// SIMATIC S7-200 project (STEP 7-Micro/WIN), CPU 226 CN REL 02.01

ORGANIZATION_BLOCK OB_1:OB1
TITLE=Ver41 add  weekly  timer  to  PLC , and  Clean Claw Pump check ;  PC program use  Ver34 edition  or  higher edition .
// Ver42  shifting  change ,  
// Ver43  add 喷雾提前结束(20060822) , PC Program 使用Ver35或以上版本
// Ver43  communication format  change  , PC程序使用Ver21或以上版本
// ver44  PC程序使用Ver21或以上版本
// Ver45  增加热补偿和PCB阻塞报警,PC程序使用Ver22或以上版本
// Ver46  增加付款条件自锁功能
// Ver47  完善喷雾（可提前或延时结束）
// ver48  细化运输模拟量参数
BEGIN
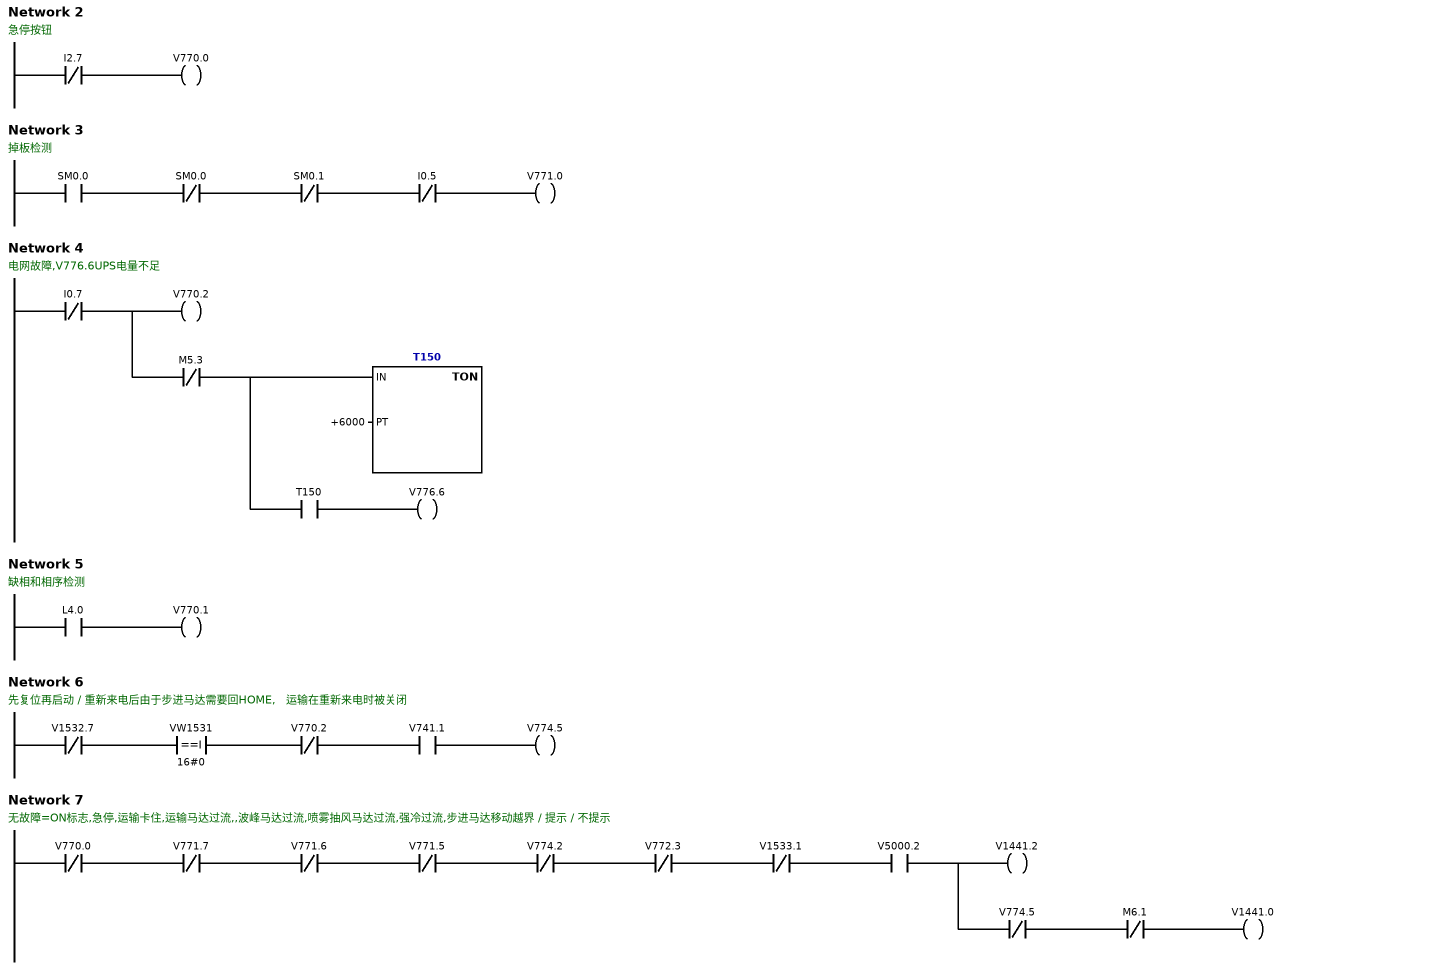
Network 2
// 急停按钮
LDN    I2.7
=      V770.0
Network 3
// 掉板检测
LD     SM0.0
AN     SM0.0
AN     SM0.1
AN     I0.5
=      V771.0
Network 4
// 电网故障,V776.6UPS电量不足
LDN    I0.7
=      V770.2
AN     M5.3
TON    T150, +6000
A      T150
=      V776.6
Network 5
// 缺相和相序检测
LD     L4.0
=      V770.1
Network 6
// 先复位再启动
// 重新来电后由于步进马达需要回HOME,   运输在重新来电时被关闭
LDN    V1532.7
AW=    VW1531, 16#0
AN     V770.2
A      V741.1
=      V774.5
Network 7
// 无故障=ON标志,急停,运输卡住,运输马达过流,,波峰马达过流,喷雾抽风马达过流,强冷过流,步进马达移动越界
// 提示
// 不提示
LDN    V770.0
AN     V771.7
AN     V771.6
AN     V771.5
AN     V774.2
AN     V772.3
AN     V1533.1
A      V5000.2
=      V1441.2
AN     V774.5
AN     M6.1
=      V1441.0
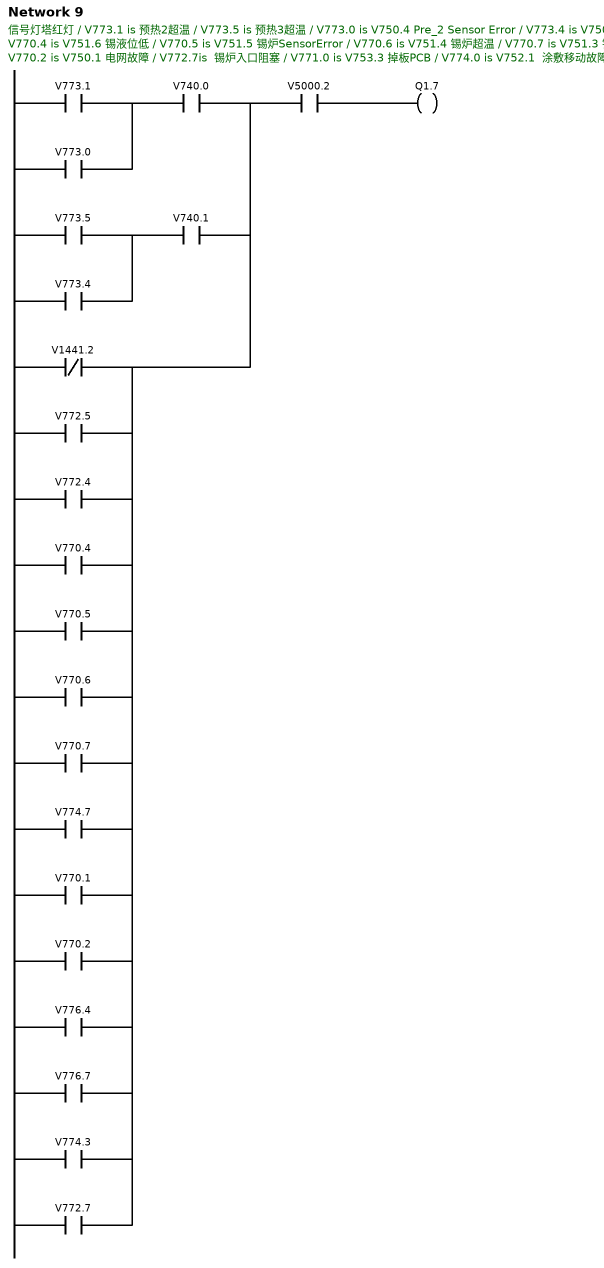
Network 9
// 信号灯塔红灯
// V773.1 is 预热2超温
// V773.5 is 预热3超温
// V773.0 is V750.4 Pre_2 Sensor Error
// V773.4 is V750.5 Pre_3 Sensor Error
// V772.5 is 预热1超温
// V772.4 is V750.3 Pre_1 Sensor Error
// 
// V770.4 is V751.6 锡液位低
// V770.5 is V751.5 锡炉SensorError
// V770.6 is V751.4 锡炉超温
// V770.7 is V751.3 锡炉参数错误
// V774.7 is V751.7  防止锡炉超温控制器
// 
// V770.1 is V750.0 电网缺相/相序错误
// V770.2 is V750.1 电网故障
// V772.7is  锡炉入口阻塞
// V771.0 is V753.3 掉板PCB
// V774.0 is V752.1  涂敷移动故障
// V776.4 is V752.3  助焊剂缺少
// V776.7 is V752.5  Clean Claw Low Limit
// V1533.1 is V752.4 步进马达移动故障
// V774.3 is V752.6 助焊剂添加故障
LD     V773.1
O      V773.0
A      V740.0
LD     V773.5
O      V773.4
A      V740.1
OLD
LDN    V1441.2
O      V772.5
O      V772.4
O      V770.4
O      V770.5
O      V770.6
O      V770.7
O      V774.7
O      V770.1
O      V770.2
O      V776.4
O      V776.7
O      V774.3
O      V772.7
OLD
A      V5000.2
=      Q1.7
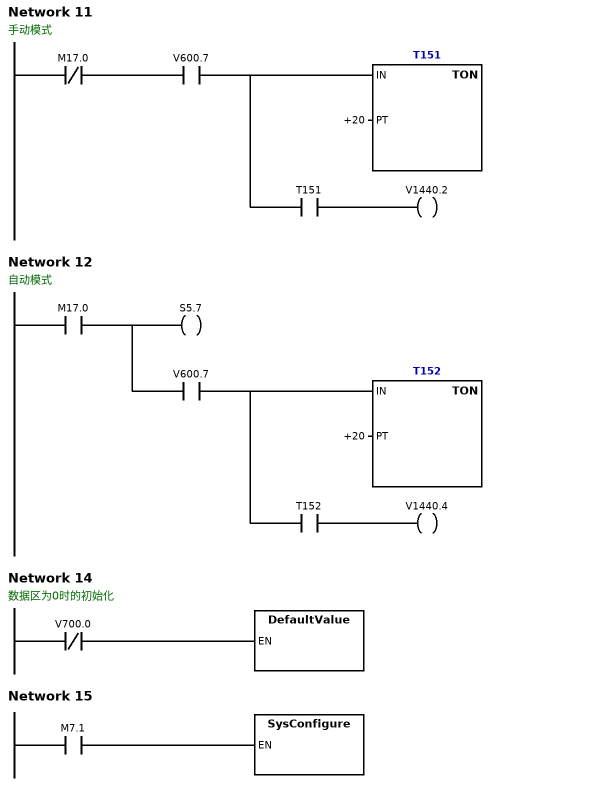
Network 11
// 手动模式
LDN    M17.0
A      V600.7
TON    T151, +20
A      T151
=      V1440.2
Network 12
// 自动模式
LD     M17.0
=      S5.7
A      V600.7
TON    T152, +20
A      T152
=      V1440.4
Network 14
// 数据区为0时的初始化
LDN    V700.0
CALL   DefaultValue:SBR18
Network 15
LD     M7.1
CALL   SysConfigure:SBR29
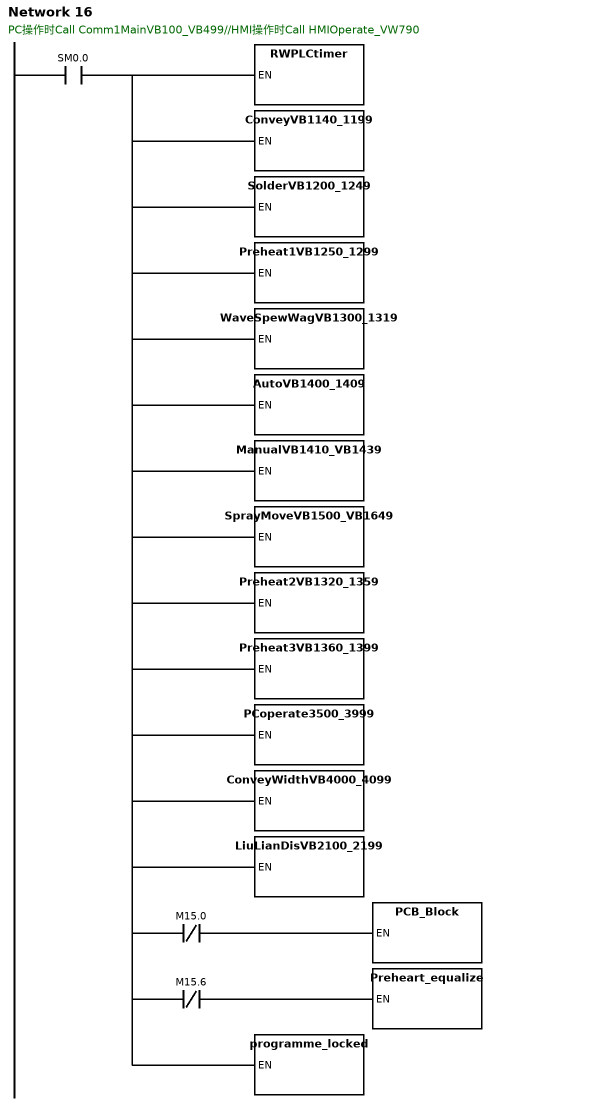
Network 16
// PC操作时Call Comm1MainVB100_VB499//HMI操作时Call HMIOperate_VW790
LD     SM0.0
LPS
CALL   RWPLCtimer:SBR1
CALL   ConveyVB1140_1199:SBR2
CALL   SolderVB1200_1249:SBR3
CALL   Preheat1VB1250_1299:SBR4
CALL   WaveSpewWagVB1300_1319:SBR5
CALL   AutoVB1400_1409:SBR8
CALL   ManualVB1410_VB1439:SBR9
CALL   SprayMoveVB1500_VB1649:SBR10
CALL   Preheat2VB1320_1359:SBR6
CALL   Preheat3VB1360_1399:SBR7
CALL   PCoperate3500_3999:SBR17
CALL   ConveyWidthVB4000_4099:SBR16
CALL   LiuLianDisVB2100_2199:SBR11
AN     M15.0
CALL   PCB_Block:SBR45
LRD
AN     M15.6
CALL   Preheart_equalize:SBR34
LPP
CALL   programme_locked:SBR46
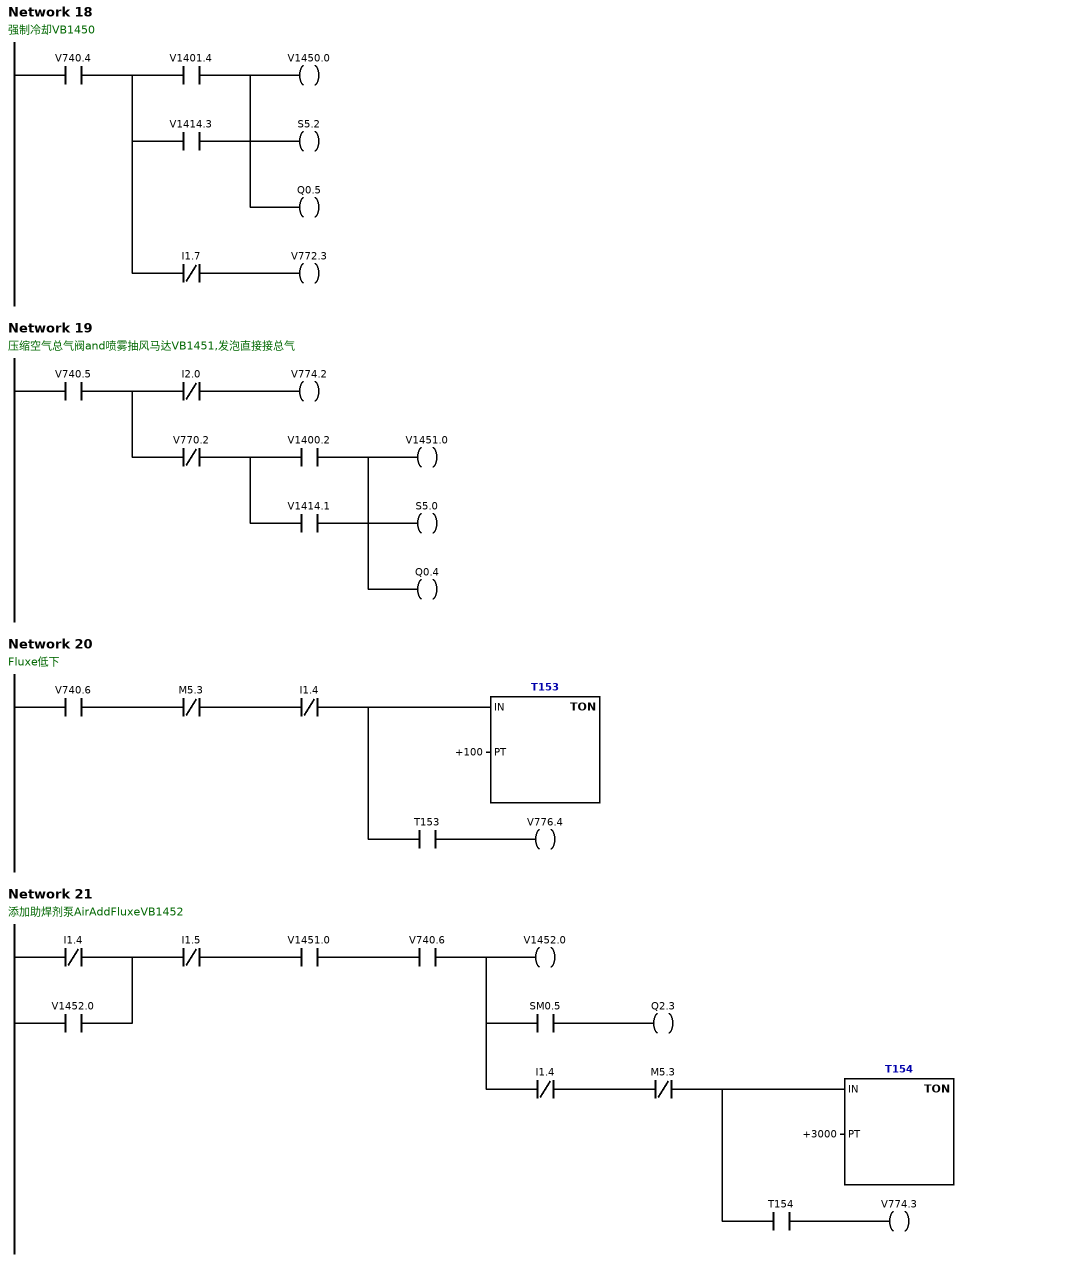
Network 18
// 强制冷却VB1450
LD     V740.4
LPS
LD     V1401.4
O      V1414.3
ALD
=      V1450.0
=      S5.2
=      Q0.5
LPP
AN     I1.7
=      V772.3
Network 19
// 压缩空气总气阀and喷雾抽风马达VB1451,发泡直接接总气
LD     V740.5
LPS
AN     I2.0
=      V774.2
LPP
AN     V770.2
LD     V1400.2
O      V1414.1
ALD
=      V1451.0
=      S5.0
=      Q0.4
Network 20
// Fluxe低下
LD     V740.6
AN     M5.3
AN     I1.4
TON    T153, +100
A      T153
=      V776.4
Network 21
// 添加助焊剂泵AirAddFluxeVB1452
LDN    I1.4
O      V1452.0
AN     I1.5
A      V1451.0
A      V740.6
LPS
=      V1452.0
A      SM0.5
=      Q2.3
LPP
AN     I1.4
AN     M5.3
TON    T154, +3000
A      T154
=      V774.3
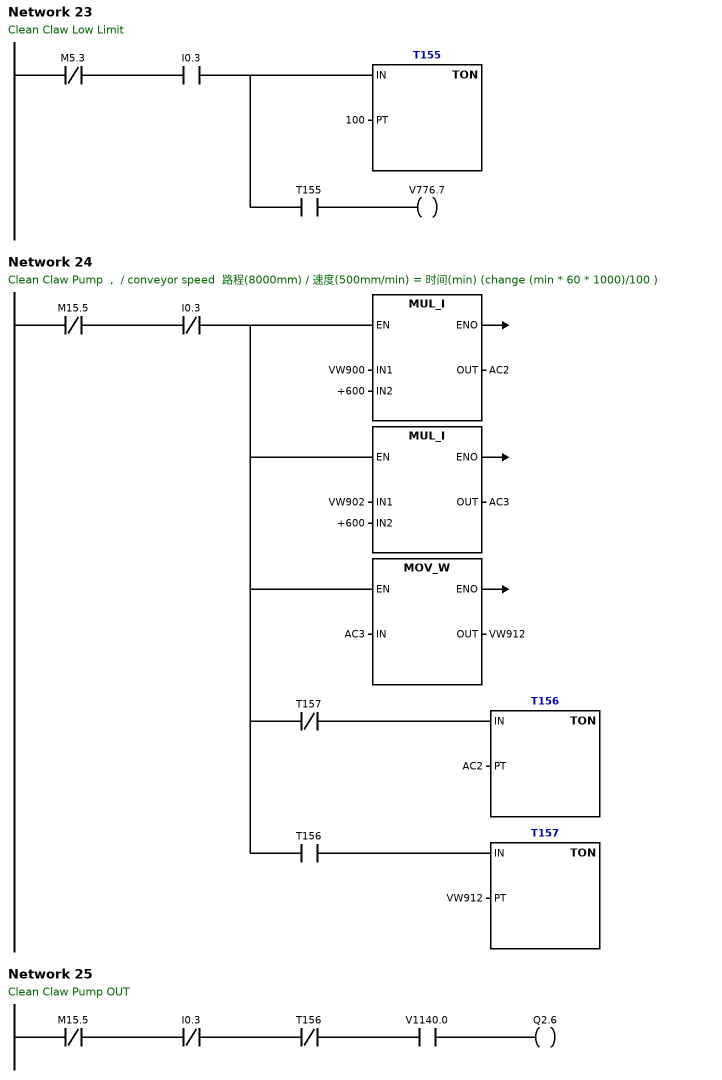
Network 23
// Clean Claw Low Limit
LDN    M5.3
A      I0.3
TON    T155, 100
A      T155
=      V776.7
Network 24
// Clean Claw Pump  , 
// conveyor speed  路程(8000mm) / 速度(500mm/min) = 时间(min) (change (min * 60 * 1000)/100 )
LDN    M15.5
AN     I0.3
LPS
MOVW   VW900, AC2
*I     +600, AC2
MOVW   VW902, AC3
*I     +600, AC3
MOVW   AC3, VW912
AN     T157
TON    T156, AC2
LPP
A      T156
TON    T157, VW912
Network 25
// Clean Claw Pump OUT
LDN    M15.5
AN     I0.3
AN     T156
A      V1140.0
=      Q2.6
END_ORGANIZATION_BLOCK

SUBROUTINE_BLOCK RWPLCtimer:SBR1
TITLE=
BEGIN
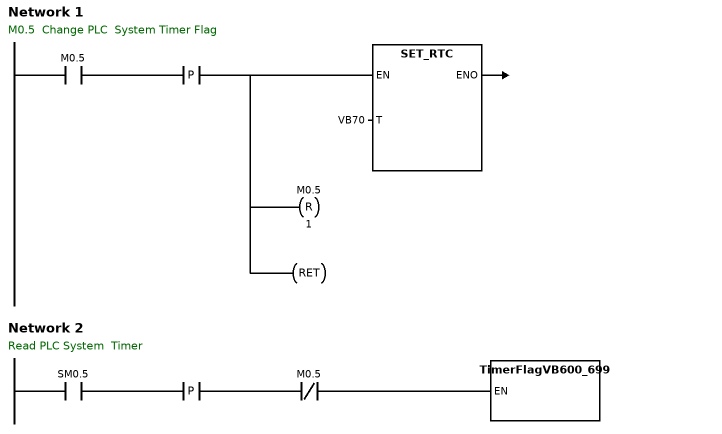
Network 1
//  M0.5  Change PLC  System Timer Flag
LD     M0.5
EU
TODW   VB70
R      M0.5, 1
CRET
Network 2 // 

// Read PLC System  Timer
LD     SM0.5
EU
AN     M0.5
CALL   TimerFlagVB600_699:SBR33
END_SUBROUTINE_BLOCK

SUBROUTINE_BLOCK ConveyVB1140_1199:SBR2
TITLE=
BEGIN
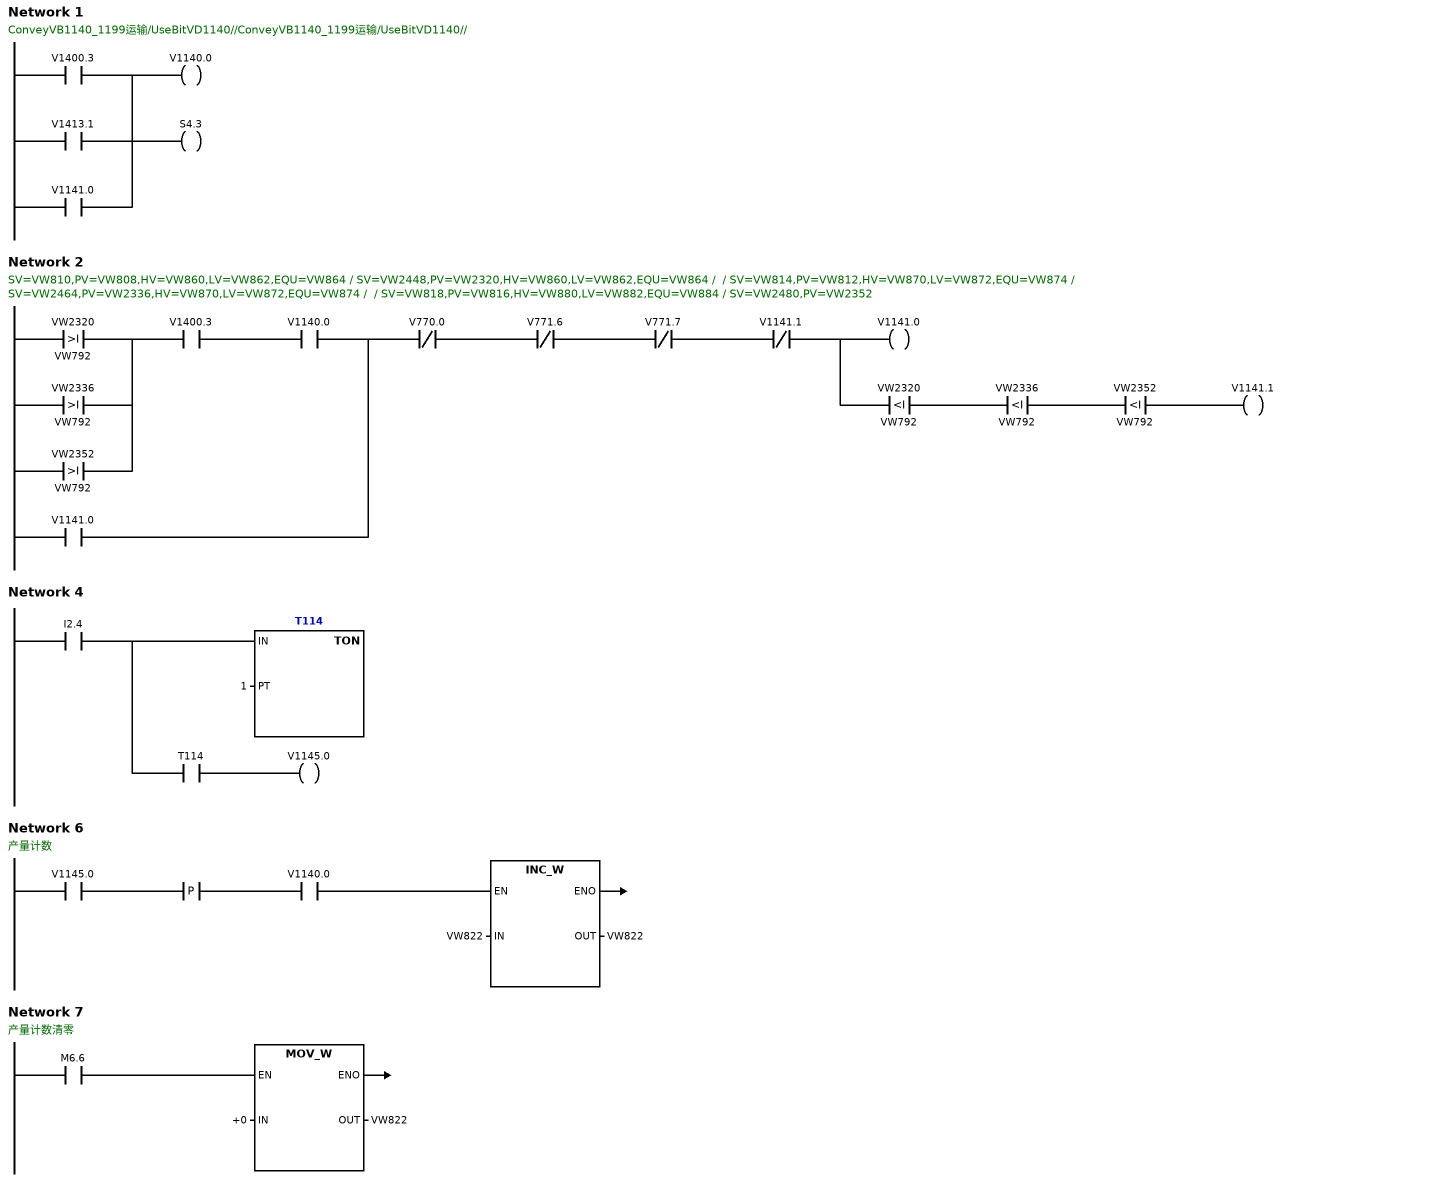
Network 1
// ConveyVB1140_1199运输/UseBitVD1140//ConveyVB1140_1199运输/UseBitVD1140//
LD     V1400.3
O      V1413.1
O      V1141.0
=      V1140.0
=      S4.3
Network 2
// SV=VW810,PV=VW808,HV=VW860,LV=VW862,EQU=VW864
// SV=VW2448,PV=VW2320,HV=VW860,LV=VW862,EQU=VW864
// 
// SV=VW814,PV=VW812,HV=VW870,LV=VW872,EQU=VW874
// SV=VW2464,PV=VW2336,HV=VW870,LV=VW872,EQU=VW874
// 
// SV=VW818,PV=VW816,HV=VW880,LV=VW882,EQU=VW884
// SV=VW2480,PV=VW2352
LDW>   VW2320, VW792
OW>    VW2336, VW792
OW>    VW2352, VW792
A      V1400.3
A      V1140.0
O      V1141.0
AN     V770.0
AN     V771.6
AN     V771.7
AN     V1141.1
=      V1141.0
AW<    VW2320, VW792
AW<    VW2336, VW792
AW<    VW2352, VW792
=      V1141.1
Network 4
LD     I2.4
TON    T114, 1
A      T114
=      V1145.0
Network 6
// 产量计数
LD     V1145.0
EU
A      V1140.0
INCW   VW822
Network 7
// 产量计数清零
LD     M6.6
MOVW   +0, VW822
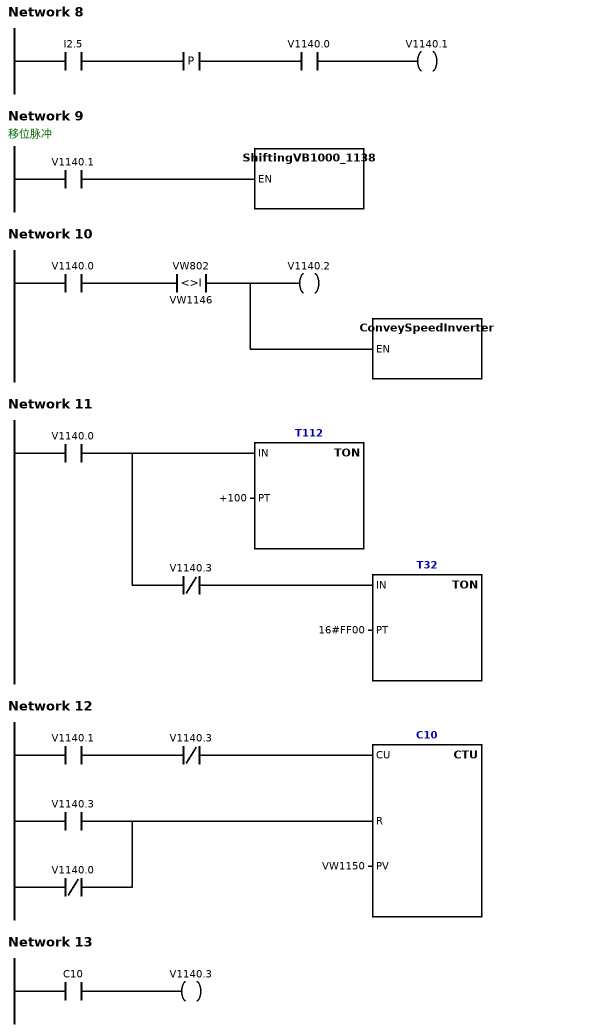
Network 8
LD     I2.5
EU
A      V1140.0
=      V1140.1
Network 9
// 移位脉冲
LD     V1140.1
CALL   ShiftingVB1000_1138:SBR19
Network 10
LD     V1140.0
AW<>   VW802, VW1146
=      V1140.2
CALL   ConveySpeedInverter:SBR20
Network 11
LD     V1140.0
TON    T112, +100
AN     V1140.3
TON    T32, 16#FF00
Network 12
LD     V1140.1
AN     V1140.3
LD     V1140.3
ON     V1140.0
CTU    C10, VW1150
Network 13
LD     C10
=      V1140.3
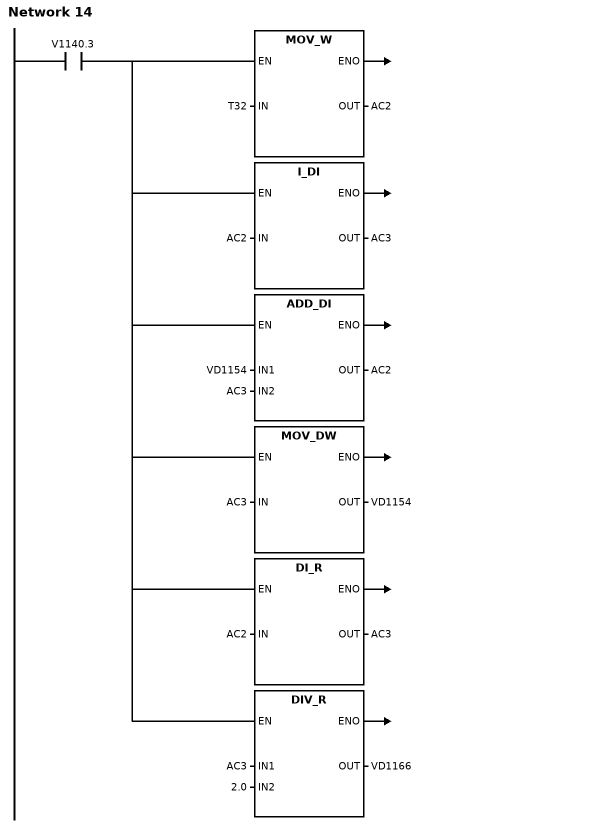
Network 14
LD     V1140.3
MOVW   T32, AC2
ITD    AC2, AC3
MOVD   VD1154, AC2
+D     AC3, AC2
MOVD   AC3, VD1154
DTR    AC2, AC3
MOVR   AC3, VD1166
/R     2.0, VD1166
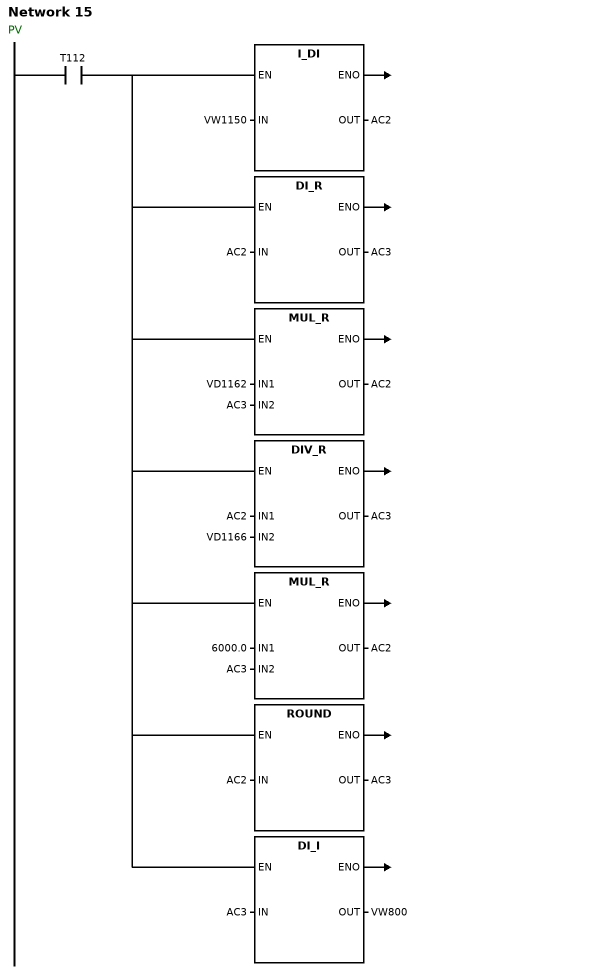
Network 15
// PV
LD     T112
ITD    VW1150, AC2
DTR    AC2, AC3
MOVR   VD1162, AC2
*R     AC3, AC2
MOVR   AC2, AC3
/R     VD1166, AC3
MOVR   6000.0, AC2
*R     AC3, AC2
ROUND  AC2, AC3
DTI    AC3, VW800
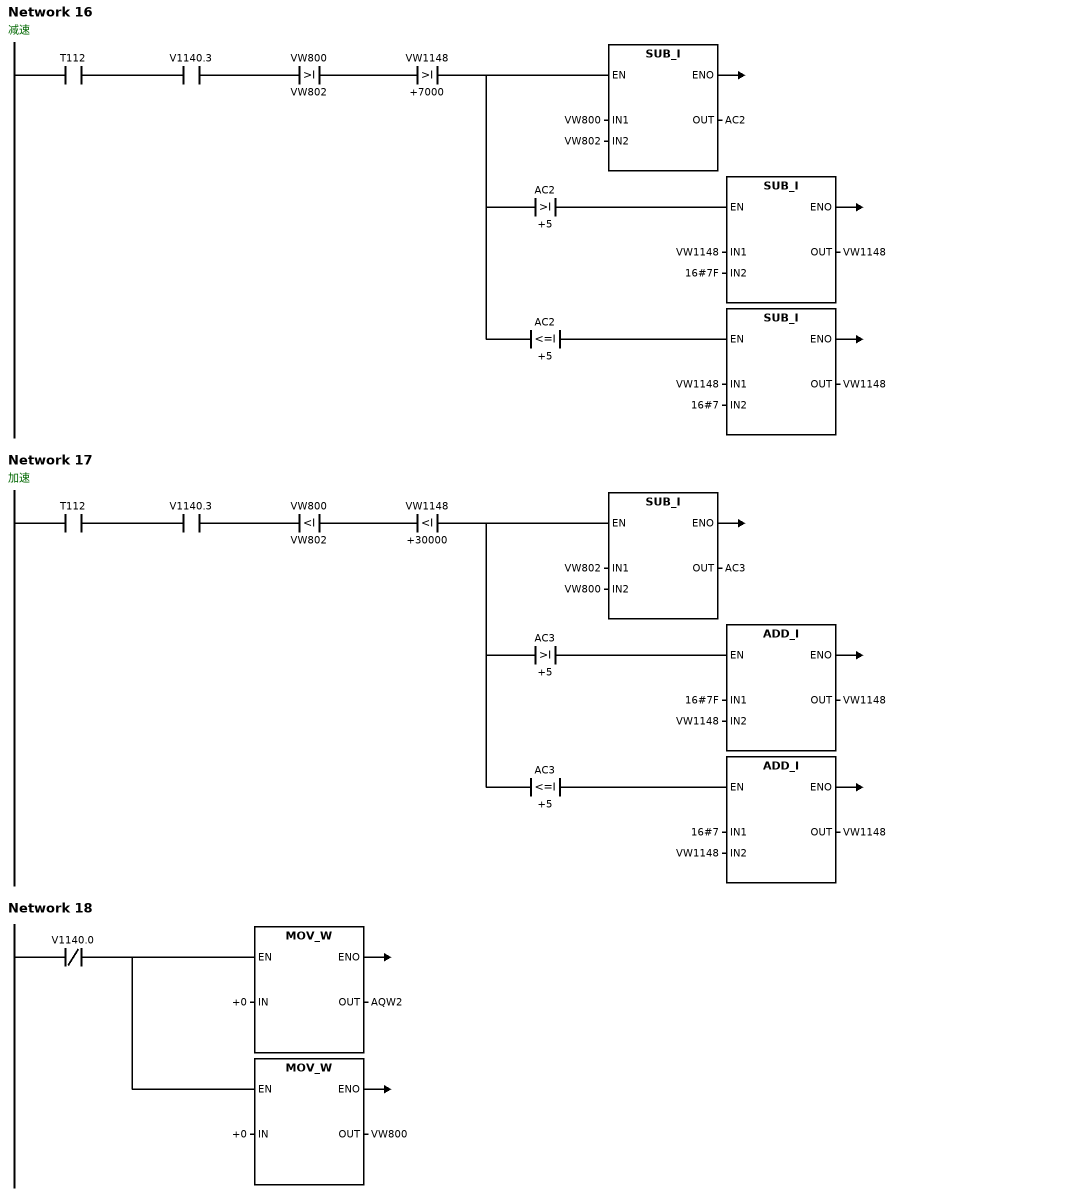
Network 16
// 减速
LD     T112
A      V1140.3
AW>    VW800, VW802
AW>    VW1148, +7000
LPS
MOVW   VW800, AC2
-I     VW802, AC2
AW>    AC2, +5
-I     16#7F, VW1148
LPP
AW<=   AC2, +5
-I     16#7, VW1148
Network 17
// 加速
LD     T112
A      V1140.3
AW<    VW800, VW802
AW<    VW1148, +30000
LPS
MOVW   VW802, AC3
-I     VW800, AC3
AW>    AC3, +5
+I     16#7F, VW1148
LPP
AW<=   AC3, +5
+I     16#7, VW1148
Network 18
LDN    V1140.0
MOVW   +0, AQW2
MOVW   +0, VW800
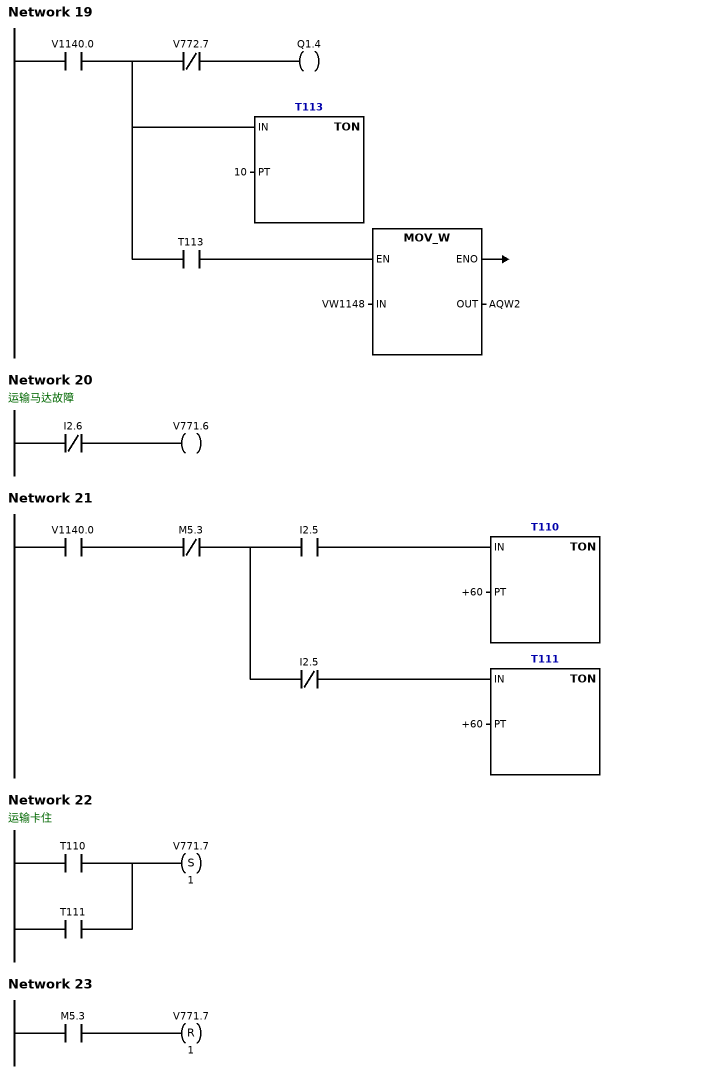
Network 19
LD     V1140.0
LPS
AN     V772.7
=      Q1.4
LRD
TON    T113, 10
LPP
A      T113
MOVW   VW1148, AQW2
Network 20
// 运输马达故障
LDN    I2.6
=      V771.6
Network 21
LD     V1140.0
AN     M5.3
LPS
A      I2.5
TON    T110, +60
LPP
AN     I2.5
TON    T111, +60
Network 22
// 运输卡住
LD     T110
O      T111
S      V771.7, 1
Network 23
LD     M5.3
R      V771.7, 1
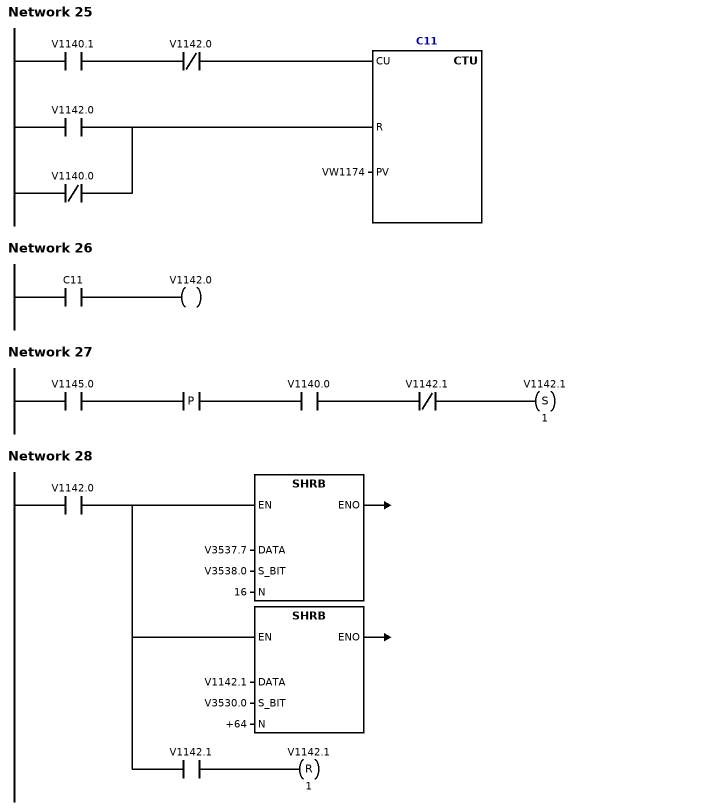
Network 25
LD     V1140.1
AN     V1142.0
LD     V1142.0
ON     V1140.0
CTU    C11, VW1174
Network 26
LD     C11
=      V1142.0
Network 27
LD     V1145.0
EU
A      V1140.0
AN     V1142.1
S      V1142.1, 1
Network 28
LD     V1142.0
SHRB   V3537.7, V3538.0, 16
SHRB   V1142.1, V3530.0, +64
A      V1142.1
R      V1142.1, 1
END_SUBROUTINE_BLOCK

SUBROUTINE_BLOCK SolderVB1200_1249:SBR3
TITLE=
BEGIN
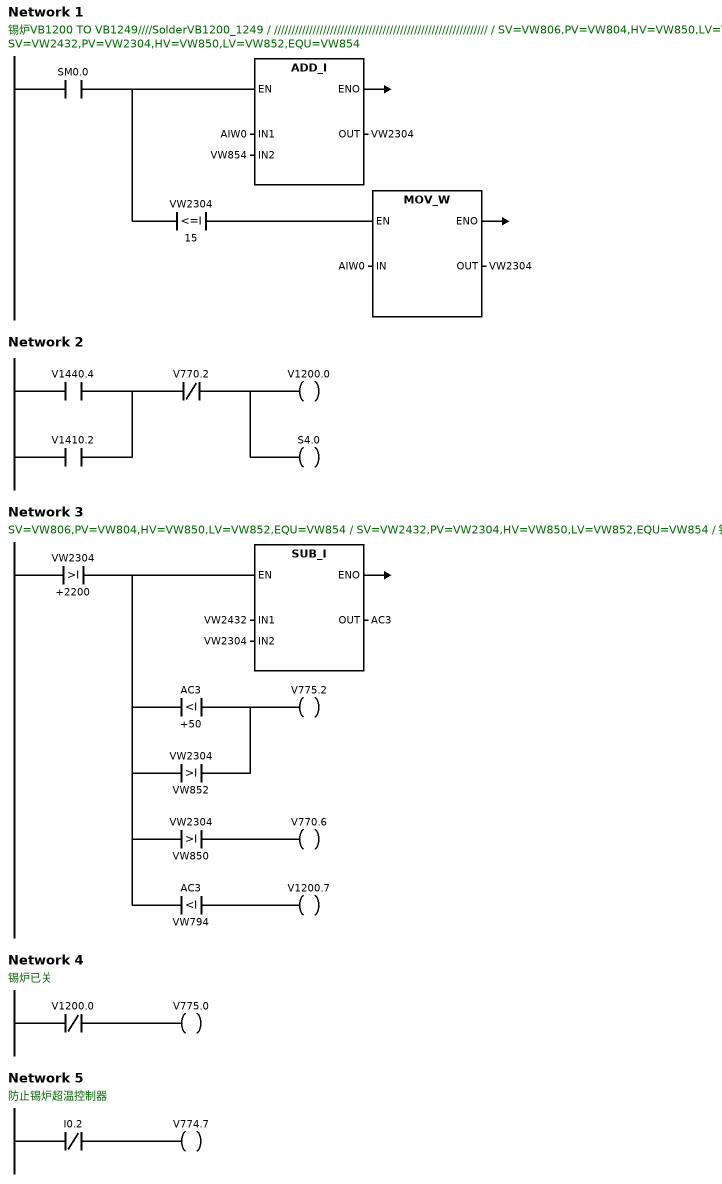
Network 1
// 锡炉VB1200 TO VB1249////SolderVB1200_1249
// /////////////////////////////////////////////////////////////
// SV=VW806,PV=VW804,HV=VW850,LV=VW852,EQU=VW854
// SV=VW2432,PV=VW2304,HV=VW850,LV=VW852,EQU=VW854
LD     SM0.0
MOVW   AIW0, VW2304
+I     VW854, VW2304
AW<=   VW2304, 15
MOVW   AIW0, VW2304
Network 2
LD     V1440.4
O      V1410.2
AN     V770.2
=      V1200.0
=      S4.0
Network 3
// SV=VW806,PV=VW804,HV=VW850,LV=VW852,EQU=VW854
// SV=VW2432,PV=VW2304,HV=VW850,LV=VW852,EQU=VW854
// 锡炉超温V770.6
// ,锡炉OK V775.2
LDW>   VW2304, +2200
LPS
MOVW   VW2432, AC3
-I     VW2304, AC3
LDW<   AC3, +50
OW>    VW2304, VW852
ALD
=      V775.2
LPP
LPS
AW>    VW2304, VW850
=      V770.6
LPP
AW<    AC3, VW794
=      V1200.7
Network 4
// 锡炉已关
LDN    V1200.0
=      V775.0
Network 5
// 防止锡炉超温控制器
LDN    I0.2
=      V774.7
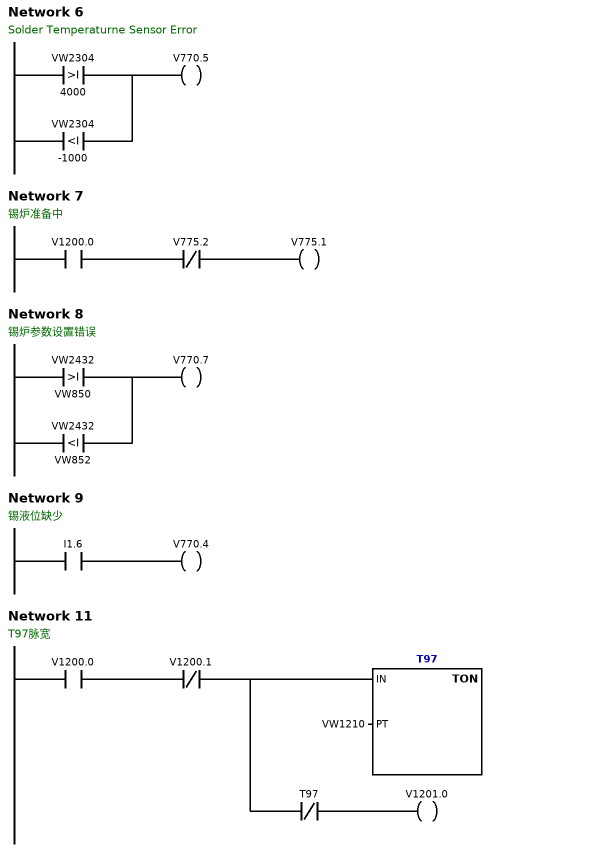
Network 6
// Solder Temperaturne Sensor Error
LDW>   VW2304, 4000
OW<    VW2304, -1000
=      V770.5
Network 7
// 锡炉准备中
LD     V1200.0
AN     V775.2
=      V775.1
Network 8
// 锡炉参数设置错误
LDW>   VW2432, VW850
OW<    VW2432, VW852
=      V770.7
Network 9
// 锡液位缺少
LD     I1.6
=      V770.4
Network 11
// T97脉宽
LD     V1200.0
AN     V1200.1
TON    T97, VW1210
AN     T97
=      V1201.0
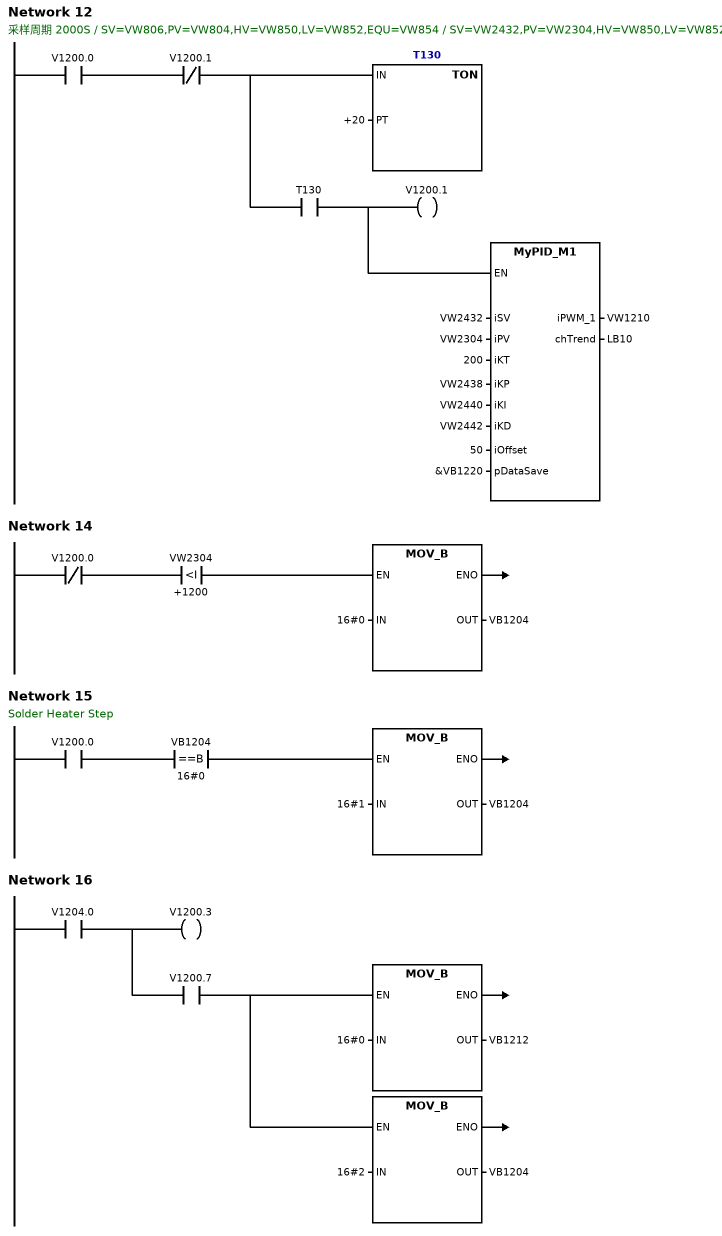
Network 12
// 采样周期 2000S
// SV=VW806,PV=VW804,HV=VW850,LV=VW852,EQU=VW854
// SV=VW2432,PV=VW2304,HV=VW850,LV=VW852,EQU=VW854
LD     V1200.0
AN     V1200.1
TON    T130, +20
A      T130
=      V1200.1
CALL   MyPID_M1:SBR30, VW2432, VW2304, 200, VW2438, VW2440, VW2442, 50, &VB1220, VW1210, LB10
Network 14
LDN    V1200.0
AW<    VW2304, +1200
MOVB   16#0, VB1204
Network 15
// Solder Heater Step
LD     V1200.0
AB=    VB1204, 16#0
MOVB   16#1, VB1204
Network 16
LD     V1204.0
=      V1200.3
A      V1200.7
MOVB   16#0, VB1212
MOVB   16#2, VB1204
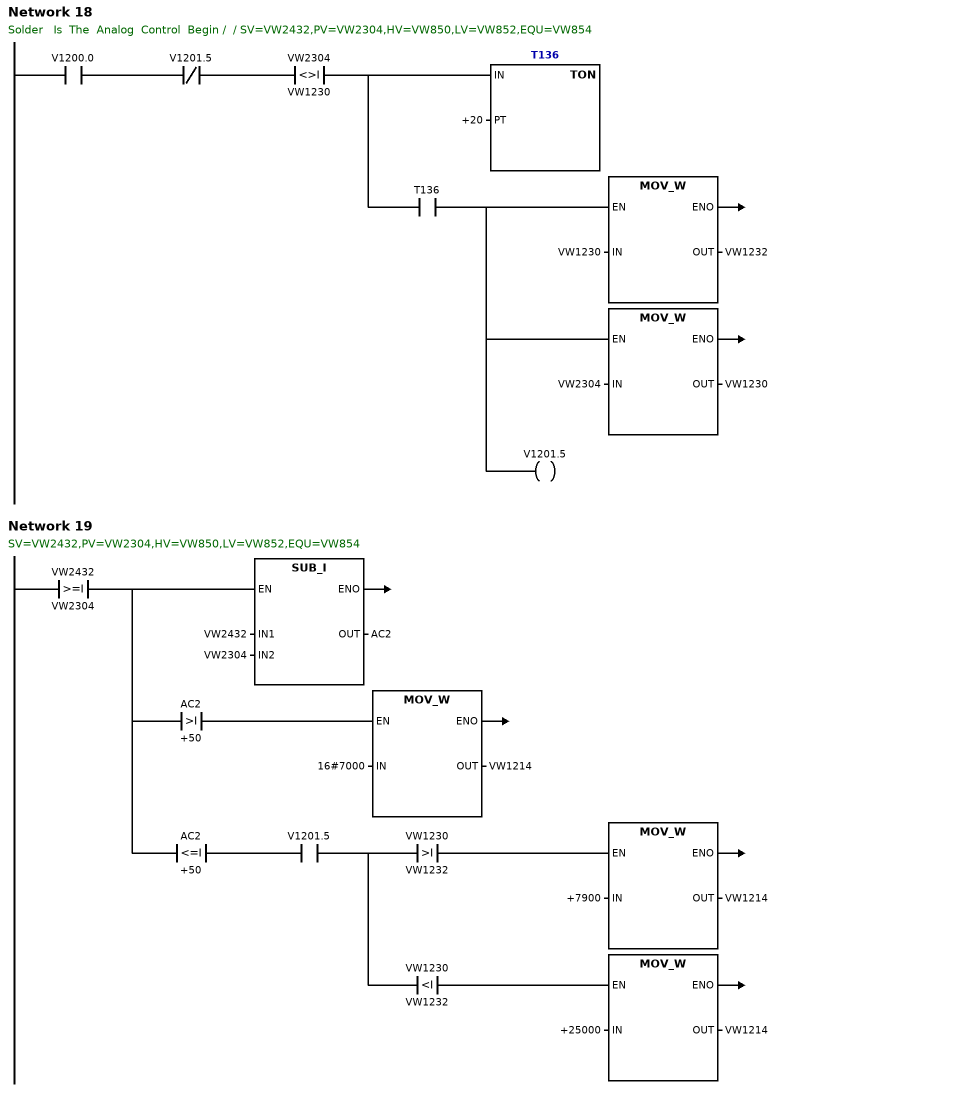
Network 18
// Solder   Is  The  Analog  Control  Begin
// 
// SV=VW2432,PV=VW2304,HV=VW850,LV=VW852,EQU=VW854
LD     V1200.0
AN     V1201.5
AW<>   VW2304, VW1230
TON    T136, +20
A      T136
MOVW   VW1230, VW1232
MOVW   VW2304, VW1230
=      V1201.5
Network 19
// SV=VW2432,PV=VW2304,HV=VW850,LV=VW852,EQU=VW854
LDW>=  VW2432, VW2304
LPS
MOVW   VW2432, AC2
-I     VW2304, AC2
AW>    AC2, +50
MOVW   16#7000, VW1214
LPP
AW<=   AC2, +50
A      V1201.5
LPS
AW>    VW1230, VW1232
MOVW   +7900, VW1214
LPP
AW<    VW1230, VW1232
MOVW   +25000, VW1214
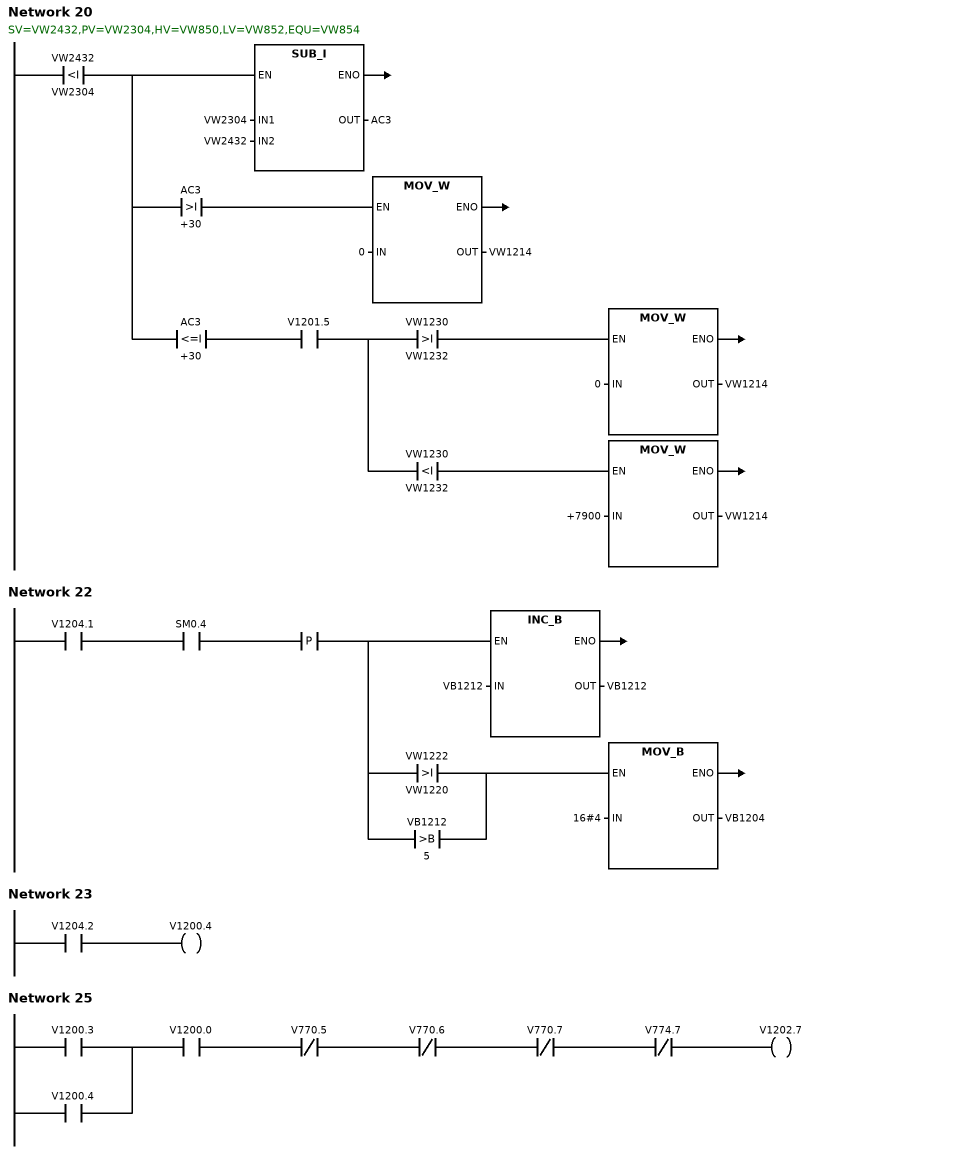
Network 20
// SV=VW2432,PV=VW2304,HV=VW850,LV=VW852,EQU=VW854
LDW<   VW2432, VW2304
LPS
MOVW   VW2304, AC3
-I     VW2432, AC3
AW>    AC3, +30
MOVW   0, VW1214
LPP
AW<=   AC3, +30
A      V1201.5
LPS
AW>    VW1230, VW1232
MOVW   0, VW1214
LPP
AW<    VW1230, VW1232
MOVW   +7900, VW1214
Network 21
// Solder   Is  The  Analog  Control  End
Network 22
LD     V1204.1
A      SM0.4
EU
INCB   VB1212
LDW>   VW1222, VW1220
OB>    VB1212, 5
ALD
MOVB   16#4, VB1204
Network 23
LD     V1204.2
=      V1200.4
Network 25
LD     V1200.3
O      V1200.4
A      V1200.0
AN     V770.5
AN     V770.6
AN     V770.7
AN     V774.7
=      V1202.7
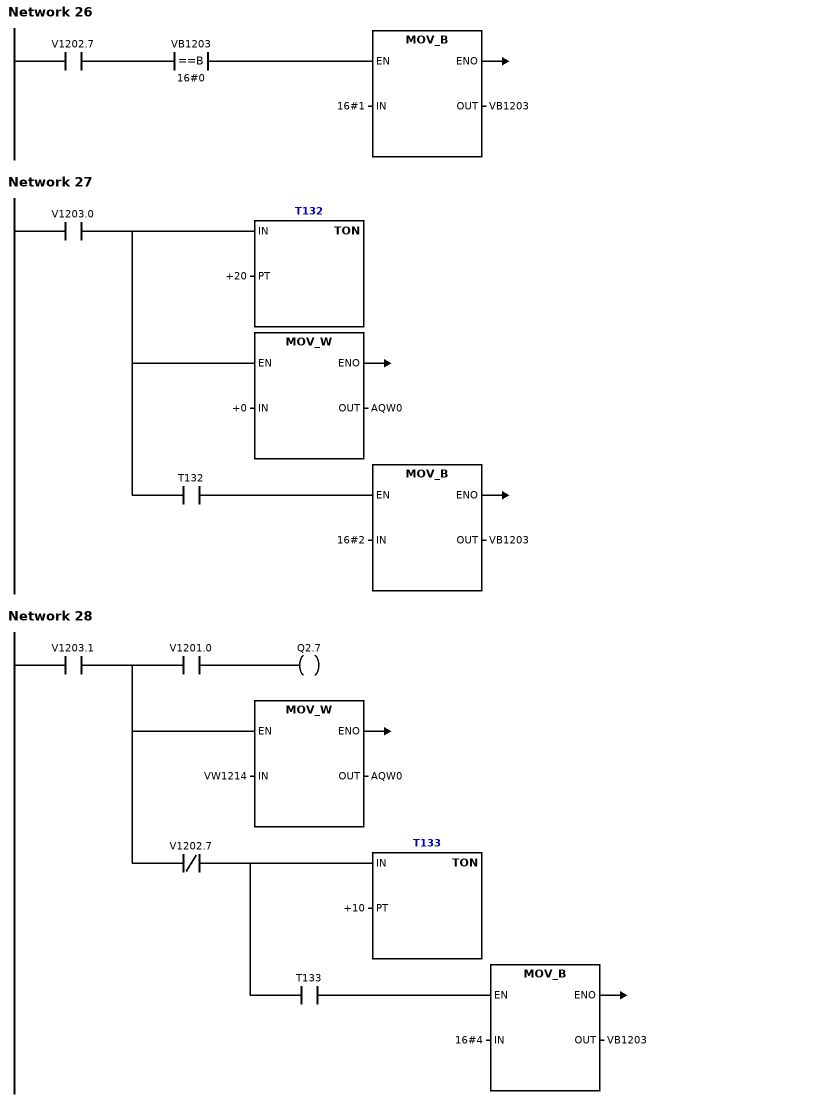
Network 26
LD     V1202.7
AB=    VB1203, 16#0
MOVB   16#1, VB1203
Network 27
LD     V1203.0
TON    T132, +20
MOVW   +0, AQW0
A      T132
MOVB   16#2, VB1203
Network 28
LD     V1203.1
LPS
A      V1201.0
=      Q2.7
LRD
MOVW   VW1214, AQW0
LPP
AN     V1202.7
TON    T133, +10
A      T133
MOVB   16#4, VB1203
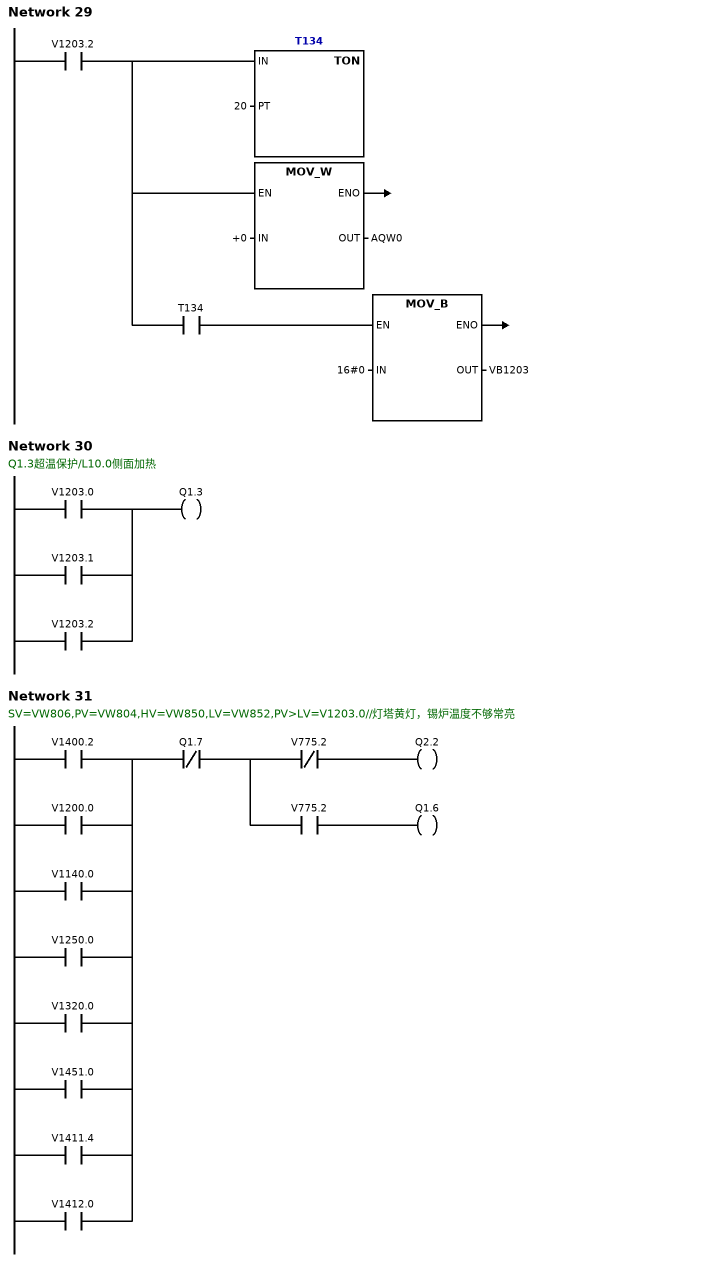
Network 29
LD     V1203.2
TON    T134, 20
MOVW   +0, AQW0
A      T134
MOVB   16#0, VB1203
Network 30
// Q1.3超温保护/L10.0侧面加热
LD     V1203.0
O      V1203.1
O      V1203.2
=      Q1.3
Network 31
// SV=VW806,PV=VW804,HV=VW850,LV=VW852,PV>LV=V1203.0//灯塔黄灯，锡炉温度不够常亮
LD     V1400.2
O      V1200.0
O      V1140.0
O      V1250.0
O      V1320.0
O      V1451.0
O      V1411.4
O      V1412.0
AN     Q1.7
LPS
AN     V775.2
=      Q2.2
LPP
A      V775.2
=      Q1.6
END_SUBROUTINE_BLOCK

SUBROUTINE_BLOCK Preheat1VB1250_1299:SBR4
TITLE=
BEGIN
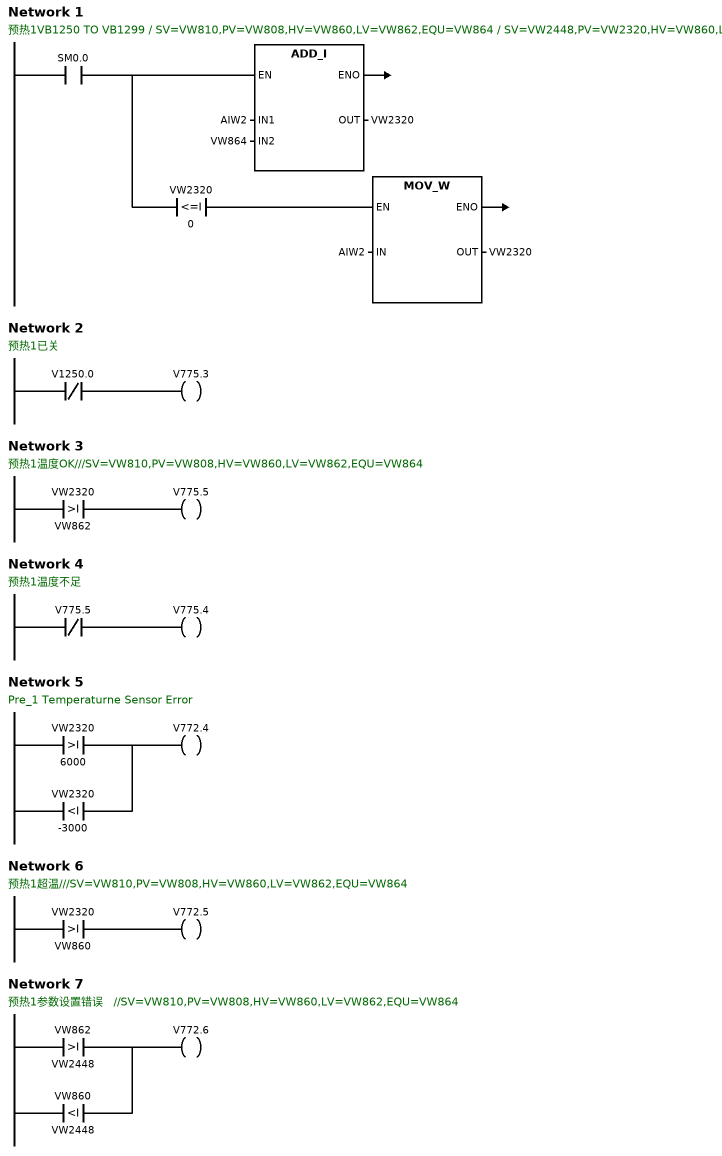
Network 1
// 预热1VB1250 TO VB1299
// SV=VW810,PV=VW808,HV=VW860,LV=VW862,EQU=VW864
// SV=VW2448,PV=VW2320,HV=VW860,LV=VW862,EQU=VW864
LD     SM0.0
MOVW   AIW2, VW2320
+I     VW864, VW2320
AW<=   VW2320, 0
MOVW   AIW2, VW2320
Network 2
// 预热1已关
LDN    V1250.0
=      V775.3
Network 3
// 预热1温度OK///SV=VW810,PV=VW808,HV=VW860,LV=VW862,EQU=VW864
LDW>   VW2320, VW862
=      V775.5
Network 4
// 预热1温度不足
LDN    V775.5
=      V775.4
Network 5
// Pre_1 Temperaturne Sensor Error
LDW>   VW2320, 6000
OW<    VW2320, -3000
=      V772.4
Network 6
// 预热1超温///SV=VW810,PV=VW808,HV=VW860,LV=VW862,EQU=VW864
LDW>   VW2320, VW860
=      V772.5
Network 7
// 预热1参数设置错误   //SV=VW810,PV=VW808,HV=VW860,LV=VW862,EQU=VW864
LDW>   VW862, VW2448
OW<    VW860, VW2448
=      V772.6
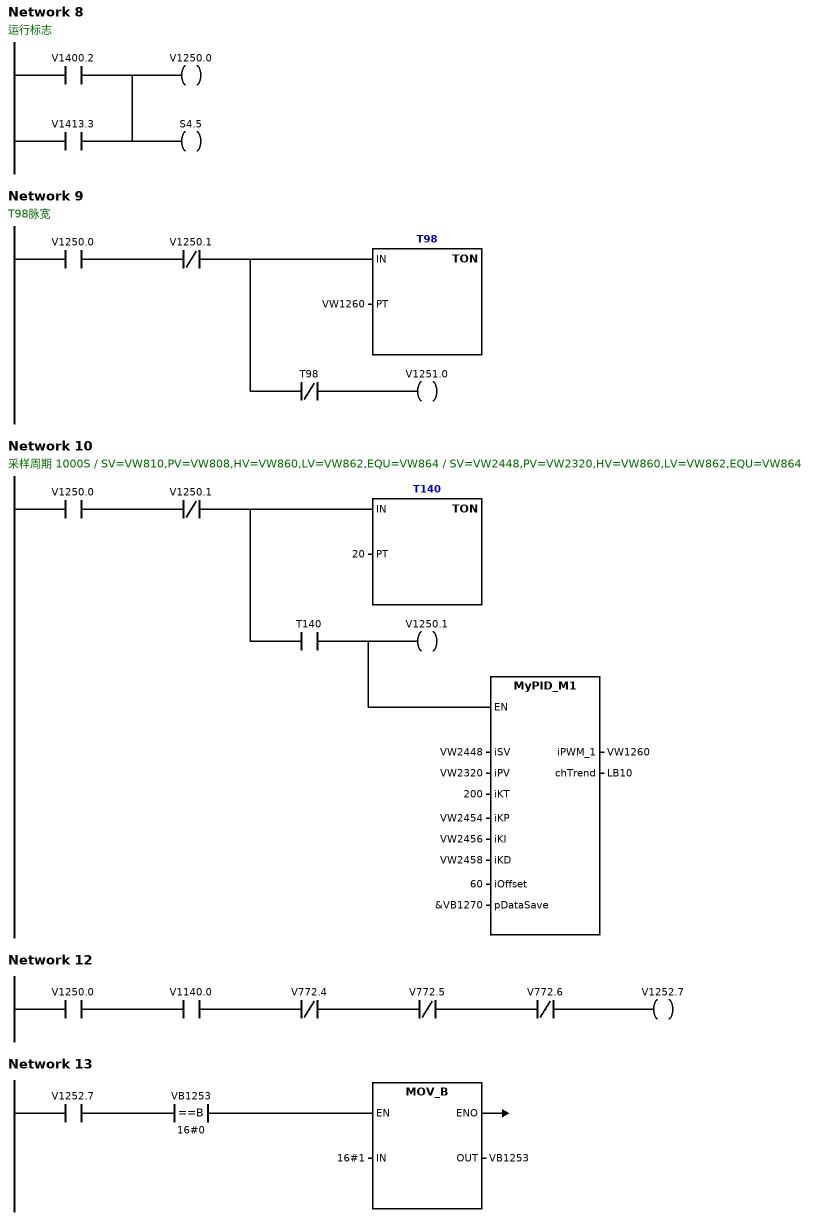
Network 8
// 运行标志
LD     V1400.2
O      V1413.3
=      V1250.0
=      S4.5
Network 9
// T98脉宽
LD     V1250.0
AN     V1250.1
TON    T98, VW1260
AN     T98
=      V1251.0
Network 10
// 采样周期 1000S
// SV=VW810,PV=VW808,HV=VW860,LV=VW862,EQU=VW864
// SV=VW2448,PV=VW2320,HV=VW860,LV=VW862,EQU=VW864
LD     V1250.0
AN     V1250.1
TON    T140, 20
A      T140
=      V1250.1
CALL   MyPID_M1:SBR30, VW2448, VW2320, 200, VW2454, VW2456, VW2458, 60, &VB1270, VW1260, LB10
Network 12
LD     V1250.0
A      V1140.0
AN     V772.4
AN     V772.5
AN     V772.6
=      V1252.7
Network 13
LD     V1252.7
AB=    VB1253, 16#0
MOVB   16#1, VB1253
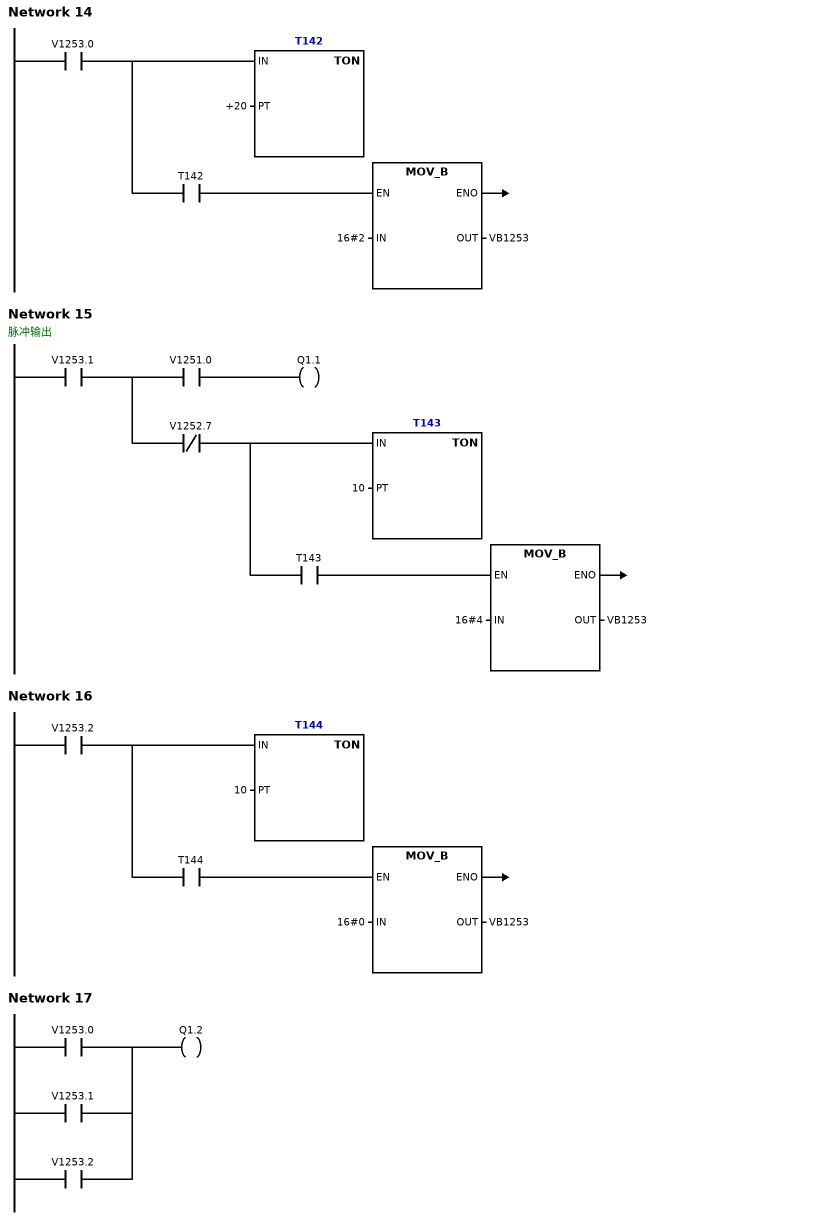
Network 14
LD     V1253.0
TON    T142, +20
A      T142
MOVB   16#2, VB1253
Network 15
// 脉冲输出
LD     V1253.1
LPS
A      V1251.0
=      Q1.1
LPP
AN     V1252.7
TON    T143, 10
A      T143
MOVB   16#4, VB1253
Network 16
LD     V1253.2
TON    T144, 10
A      T144
MOVB   16#0, VB1253
Network 17
LD     V1253.0
O      V1253.1
O      V1253.2
=      Q1.2
